TYPE (* A Structure with 2 BYTES *)
  (* Version 1.0, 2024-02-21, Franz Höpfinger, HR Agrartechnik GmbH *)
  PACKAGE logiBUS::utils::conversion::types;
  ST02B : STRUCT
    B_00 : BYTE; (* BYTE 00 *)
    B_01 : BYTE; (* BYTE 01 *)
  END_STRUCT;
END_TYPE
